TYPE EOAT :
STRUCT
	id : SectionEnum;
	material : STRING;
END_STRUCT
END_TYPE

(* stored: Version 1.1.0.1, ProductVersion 3.1.4024.11
   DUT EOAT: Id {f0393144-bb2d-431b-8fc8-9ee9221bb18e} *)
